// TIA Portal V17 export
// export: Created 2024-09-02T12:49:58.9546289Z, ExportSetting WithDefaults, DisplayName Totally Integrated Automation Portal, DisplayVersion V17, DisplayName TIA Portal Openness, DisplayVersion V17, DisplayName TIA Portal Version Control Interface, DisplayVersion V17, DisplayName STEP 7 Professional, DisplayVersion V17, DisplayName STEP 7 Safety, DisplayVersion V17, DisplayName WinCC Professional, DisplayVersion V17
DATA_BLOCK "LTLL_EE"   // DB10
TITLE = LTLL_EE
{ S7_Optimized_Access := 'FALSE'; DB_Accessible_From_OPC_UA := 'FALSE' }
AUTHOR : Siemens
FAMILY : HMI_Lite
NAME : LTLL_EE
VERSION : 8.10
// stored: AutoNumber true, DBAccessibleFromOPCUA false, InstanceOfName LTLL_typeEE, InstanceOfType UDT, IsOnlyStoredInLoadMemory false, IsWriteProtectedInAS false
"LTLL_typeEE"
   // VAR
   //    operationSeqEquipment : String[10];
   //    inventoryNumber : String[20];
   //    minMeasurementTimeActual : Time;
   //    minMeasurementTimeTarget : Time;
   //    numberOfCyclesActual : DWord;
   //    numberOfCyclesTarget : DWord;
   //    lastReset : Date_And_Time;
   //    numberOfPartsMeasurement : DWord;
   //    numberOfPartsSinceReset : DWord;
   //    totalWorkpieceCounter : DWord;
   //    numberForAlarm : Byte;
   //    totalReset : Bool;
   //    measurementStop : Bool;
   //    measurementStart : Bool;
   //    setpointsShow : Bool;
   //    offExceed : Bool;
   //    standbyExceed : Bool;
   //    operationalExceed : Bool;
   //    workingExceed : Bool;
   //    powerupExceed : Bool;
   //    powerdownExceed : Bool;
   //    reserved00 : Bool;
   //    reserved01 : Bool;
   //    reserved02 : Bool;
   //    reserved03 : Bool;
   //    reserved04 : Bool;
   //    reserved05 : Bool;
   //    energyTypes { S7_SetPoint := 'True'} : Array[0..19] of "LTLL_typeEnergyType";
   // END_VAR
BEGIN
END_DATA_BLOCK
